// Write Only Decorator for function blocks that impliment I_List interface
{attribute 'enable_dynamic_creation'}
FUNCTION_BLOCK FB_Write_Only_List EXTENDS FB_Collection IMPLEMENTS I_Write_Only_List
VAR_INPUT
	ipList : I_List;
END_VAR

(* Returns -1 as this is a write-only list *)
PROPERTY _Count : DINT
GET
_Count := -1;
END_GET
END_PROPERTY

PROPERTY _Error_Status : ST_ERROR
GET
IF THIS^.NullReferenceException() THEN _Error_Status := THIS^.stError; RETURN; END_IF
THIS^.stError := THIS^.ipList._Error_Status;
_Error_Status := F_Error(THIS^.stError.bSTATUS, THIS^.stError.nCODE, THIS^.stError.sSOURCE);
END_GET
END_PROPERTY

(* Returns FALSE as this is a write-only list *)
PROPERTY _Is_Empty : BOOL
GET
END_GET
END_PROPERTY

// Adds an item to the end of the list
METHOD Add_Back : I_Write_Only_List
VAR_INPUT
	Item 	: ANY; // Value to store in list
END_VAR
VAR_OUTPUT
	bSuccess : BOOL;
END_VAR
Add_Back := THIS^;
IF THIS^.NullReferenceException() THEN RETURN; END_IF
THIS^.ipList.Add_Back(Item, bSuccess => bSuccess);
END_METHOD

// Adds an item at the front of the list
METHOD Add_Front : I_Write_Only_List
VAR_INPUT
	Item 	: ANY; // Value to store in list
END_VAR
VAR_OUTPUT
	bSuccess : BOOL;
END_VAR
Add_Front := THIS^;
IF THIS^.NullReferenceException() THEN RETURN; END_IF
THIS^.ipList.Add_Front(Item, bSuccess => bSuccess);
END_METHOD

// Empties/Clears/Deletes every item in the collection
METHOD Clear
IF THIS^.NullReferenceException() THEN RETURN; END_IF
THIS^.ipList.Clear();
END_METHOD

// Adds new item to list at specified location, if index = 0, item will be added at the front, if index = count, item will be added at the back
METHOD Insert : I_Write_Only_List
VAR_INPUT
	Item 	: ANY;  // Item to store in list
	nIndex 	: DINT; // Location of item
END_VAR
VAR_OUTPUT
	bSuccess : BOOL;
END_VAR
Insert := THIS^;
IF THIS^.NullReferenceException() THEN RETURN; END_IF
THIS^.ipList.Insert(Item, nIndex, bSuccess => bSuccess);
END_METHOD

METHOD PROTECTED NullReferenceException : BOOL
NullReferenceException := THIS^.ipList = 0;
IF NOT NullReferenceException THEN RETURN; END_IF
THIS^.RaiseException(2000+GVL_CmpErrors.ERR_INVALID_REFERENCE, 'Null or Invalid Reference');
END_METHOD

// Removes item at the front of the list and returns nothing
METHOD Remove : I_Write_Only_List
VAR_OUTPUT
	bSuccess : BOOL;
END_VAR
Remove := THIS^;
IF THIS^.NullReferenceException() THEN RETURN; END_IF
THIS^.ipList.Remove(bSuccess => bSuccess);
END_METHOD

// Remove item at specified location and return nothing
METHOD Remove_At : I_Write_Only_List
VAR_INPUT
	nIndex : DINT; // Location of item
END_VAR
VAR_OUTPUT
	bSuccess : BOOL;
END_VAR
Remove_At := THIS^;
IF THIS^.NullReferenceException() THEN RETURN; END_IF
THIS^.ipList.Remove_At(nIndex, bSuccess => bSuccess);
END_METHOD

// Removes item at the back of the list and returns nothing
METHOD Remove_Last : I_Write_Only_List
VAR_OUTPUT
	bSuccess : BOOL;
END_VAR
Remove_At := THIS^;
IF THIS^.NullReferenceException() THEN RETURN; END_IF
THIS^.ipList.Remove_Last(bSuccess => bSuccess);
END_METHOD

// Manually resize list. If list becomes smaller, item on higher locations will be deleted.
METHOD Resize : I_Write_Only_List
VAR_INPUT
	nSize : DINT; // New size of list.
END_VAR
VAR_OUTPUT
	bSuccess : BOOL;
END_VAR
Resize := THIS^;
IF THIS^.NullReferenceException() THEN RETURN; END_IF
THIS^.ipList.Resize(nSize, bSuccess => bSuccess);
END_METHOD

// Reverses the order of items in the list
METHOD Reverse : I_Write_Only_List
VAR_OUTPUT
	bSuccess : BOOL;
END_VAR
Reverse := THIS^;
IF THIS^.NullReferenceException() THEN RETURN; END_IF
THIS^.ipList.Reverse(bSuccess => bSuccess);
END_METHOD

// Adds new item to list in the specified location without resizing list
METHOD Set : I_Write_Only_List
VAR_INPUT
	Item 	: ANY; 	// Item to store in list
	nIndex 	: DINT; // Location of item
END_VAR
VAR_OUTPUT
	bSuccess : BOOL;
END_VAR
Set := THIS^;
IF THIS^.NullReferenceException() THEN RETURN; END_IF
THIS^.ipList.Set(Item, nIndex, bSuccess => bSuccess);
END_METHOD

END_FUNCTION_BLOCK

(* stored: Version 1.1.0.1, ProductVersion 3.1.4024.4
   POU FB_Write_Only_List: Id {9182d7fd-2644-409c-aff4-167d0ab978b1}, SpecialFunc None
   Folder Exceptions: Id {01d7a93f-fb56-4c69-8936-09e6e6191e3a}
   Property _Count: Id {d81641b8-5c3f-41ed-badb-e64d206ece05}
   Get Get: Id {1fa8f3c7-35b4-4e9f-9392-3926d8db2183}
   Property _Error_Status: Id {dcc24c06-d0fb-4a70-8a55-79a0db0b534a}
   Get Get: Id {d66d964f-fa89-42f4-ba95-5bfddcdd74dc}
   Property _Is_Empty: Id {8e9c2b64-8b9b-4160-bcb2-daead2934376}
   Get Get: Id {628a248f-2051-4a66-85bd-cc4c1b574b10}
   Method Add_Back: Id {7b1287dd-2649-4f81-b964-65c5ab2ce4d7}
   Method Add_Front: Id {c90da460-4c32-4440-8eaf-1787eb5245b2}
   Method Clear: Id {25a73d91-decc-40f5-81fc-00c740294cad}
   Method Insert: Id {6d18b440-9b80-4187-8faf-ffc2e2589f41}
   Method NullReferenceException: Id {9eb3fe3d-fecc-4438-8ca2-f8de9026581a}
   Method Remove: Id {27b4e4aa-1fac-46f6-b798-41fd8ac325ca}
   Method Remove_At: Id {c9825f5a-49c3-43de-8809-6a69f087b470}
   Method Remove_Last: Id {02f897ad-59fd-4638-8df2-fd17501bfc1b}
   Method Resize: Id {e0898826-de81-4247-8142-cb664c9b3513}
   Method Reverse: Id {eeadd024-e87a-45ba-aca1-413a48293c8a}
   Method Set: Id {7820293c-2f16-4c4e-bb78-4df04964fd16} *)
